(* IEC 61131-3 sources: CodesysTest/alpha/export (part 5) *)

(* ---- MotorizedSealFlattenersFB.st ---- *)
FUNCTION_BLOCK MotorizedSealFlattenersFB EXTENDS BaseComponentFB IMPLEMENTS IComponentStatus
VAR_INPUT
    {warning 'TODO: Make a struct for some of these - too many inputs'}
	sealFlattenersVerticalAxis : ICylinder();
    clearanceOffset : REAL := 0.75;        // Clearance Offset in inches
    inSetpoint : REAL := 1.25;            // In setpoint in inches
    outSetpoint : REAL := 17.7;            // Out (sealing) setpoint in inches
    bagHoldingSetpoint : REAL := 17;    // Bag holding setpoint in inches
    clearanceSpeed : INT := 3000;        // Speed to move in clearance move
    moveInSpeed : INT := 3000;            // Speed to move in in move
    moveOutSpeed : INT := 1000;            // Speed to move in out move
    moveBagHoldingSpeed : INT := 10000;    // Speed to move in bag holding move
    fingersUpSetpoint : REAL := 0;     // Fingers Up setpoint in inches
    fingersDownSetpoint : REAL := 1.1; // Fingers down setpoint in inches
    moveFingersSpeed : INT := 2000;        // Speed to move fingers
    horizontalAxisAccel : INT := 1000;    // Accel setpoint for horizontal axis
    horizontalAxisDecel : INT := 1000;    // Decel Setpoint for horizontal axis
    verticalAxisAccel : INT := 150;    // Accel setpoint for vertical axis
    verticalAxisDecel : INT := 150;    // Decel Setpoint for vertical axis
    testMovePB : BOOL;
    testMoveSP : REAL;
    stopPB : BOOL;
    startPB : BOOL;
    nextSeqPB : BOOL;
    delay : TON := (PT:= T#300MS);
	fingersDownDelay : Standard.TON := (PT := T#200MS);

	manualPosSetpoint : REAL;

END_VAR
VAR_IN_OUT
	jogIn : BOOL;
	jogOut : BOOL;
	raiseService : BOOL;
	lowerService : BOOL;
	moveToManualSetpoint : BOOL;
END_VAR
VAR_OUTPUT
    state : SEAL_FLATTENER_STATES;
END_VAR
VAR
    //pressureBarMotor : FB_FestoMotor();
    //sealFlattenersVerticalAxisMotor : FB_AppliedMotionStepServoRTU();
	jogInONS: FB_ONS;
	jogOutONS: FB_ONS;
	jogSpeed : INT := 100;
    sealFlattenersHorizontalAxisMotor : FB_AppliedMotionStepServoEIPBaseQX();
	defaultCurrentMSF : DINT := 150;
	outCurrentMSF : DINT := 150;
	bagHoldingCurrentMSF : DINT := 85;
    enableMotorizedSealFlattenersONS : R_TRIG();
    _amMoveOut : BOOL;                // Auto mode move out command
	_amMoveIn : BOOL;
    _amMoveClearance : BOOL;            // Auto mode move Clearance command
    _amMoveInToBagHolding : BOOL;    // Auto mode move in then bag holding command
END_VAR

//    Function Block:  MotorizedSealFlattenersFB
//    Description: State machine and motor management for motorized seal flateners
//    Currently, this code requires one to use the Oriental drive with pre-programmed
//    sequence for the horizontal axis
//    Created by: Ben Hess
//    Created Date: Friday, April 6, 2018
SUPER^();
// Setup and execute 2 motor axis'

// Temporary delay between states for testing
fingersDownDelay();
delay();
jogInONS(CLK := jogIn);
jogOutONS(CLK := jogOut);
IF autoModeSelected THEN
    delay.PT := T#300MS;
ELSE
    delay.PT := T#750MS;
END_IF

outSetpoint := HMIData.bagWidth + 0.2;
bagHoldingSetpoint := HMIData.bagWidth;

// Setup the vertical axis motor
sealFlattenersVerticalAxis.Execute();

// Setup the horizontal axis motor
(*
sealFlattenersHorizontalAxisMotor(modbusInBuffer := OrientalMotorModbusRead,
                stepsPerInchSetpoint := 125,
                reversePolarity := FALSE,
                operatingCurrentDefault := 500,
                modbusCommandOutBuffer := OrientalMotorCommandWrites,
                modbusParametersOutBuffer := OrientalMotorParameterWrites,
                triggerCommandWrite => OrientalMotorTriggerCommandWrite,
                triggerParameterWrite => OrientalMotorTriggerParameterWrite);
sealFlattenersHorizontalAxisMotor.Execute();
*)

sealFlattenersHorizontalAxisMotor(ptrEIPInputs := ADR(sealFlattenerHorizontalMotorInputs),
                ptrEIPOutputs := ADR(sealFlattenerHorizontalMotorOutputs),
                stepsPerInchSetpoint := Globals.STEPS_PER_INCH_SEAL_FLATTENER_HORIZONTAL_AXIS_MOTOR,
                faultHandler := PRG_Bagger.faultHandler,
				reversePolarity := TRUE,
				defaultCurrentSetpoint := defaultCurrentMSF,
				commFail := MSFMotor.udiState <> 4,
				isHomable := TRUE);

sealFlattenersHorizontalAxisMotor.Execute();

//Report as ready if mode is auto and we're not faulted
_ready := (_mode = DEVICE_MODES.Auto) AND NOT (state = SEAL_FLATTENER_STATES.Fault);

enableMotorizedSealFlattenersONS(CLK := enable);
IF stopPB THEN
    sealFlattenersHorizontalAxisMotor.Stop();
    stopPB := FALSE;
END_IF

IF startPB AND semiAutoModeSelected THEN
    //sealFlattenersHorizontalAxisMotor.StartOperation();
    startPB := FALSE;
END_IF

IF nextSeqPB THEN
    //sealFlattenersHorizontalAxisMotor.NextSequence();
    nextSeqPB := FALSE;
END_IF

IF testMovePB THEN
    sealFlattenersHorizontalAxisMotor.MoveToPosition(position := (testMoveSP), acceleration := 100, deceleration := 100, velocity := 600);
    testMovePB := FALSE;
END_IF

IF enableONS.Q OR resetONS.Q THEN
    state := SEAL_FLATTENER_STATES.Idle;
	sealFlattenersHorizontalAxisMotor.Reset();
	_reset := FALSE;
	ClearCommands();
END_IF

IF NOT enable THEN
    state := SEAL_FLATTENER_STATES.Fault;
END_IF

// State amchine for motorized seal flatteners
CASE state OF

    SEAL_FLATTENER_STATES.Idle :                                    //If enabled move to out
                                                                    IF enable AND semiAutoModeSelected OR (autoModeSelected AND _amMoveOut) THEN
                                                                        state := SEAL_FLATTENER_STATES.MoveFlattenersOut;
                                                                        ClearCommands();
                                                                    END_IF

																	IF enable AND autoModeSelected AND _amMoveIn OR _amMoveInToBagHolding THEN
																	//IF enable AND autoModeSelected AND _amMoveIn THEN
																		sealFlattenersVerticalAxis.Retract();
																		state := SEAL_FLATTENER_STATES.MoveFlattenersIn;
																		ClearCommands();
																	END_IF

																	IF jogInONS.OSR THEN
																		sealFlattenersHorizontalAxisMotor.MoveDistance(distance := -18,
																									acceleration := horizontalAxisAccel,
																									deceleration := horizontalAxisDecel,
																									velocity := jogSpeed);
																	ELSIF jogOutONS.OSR THEN
																		sealFlattenersHorizontalAxisMotor.MoveDistance(distance := 18,
																									acceleration := horizontalAxisAccel,
																									deceleration := horizontalAxisDecel,
																									velocity := jogSpeed);
																	ELSIF jogInONS.OSF OR jogOutONS.OSF THEN
																		sealFlattenersHorizontalAxisMotor.Stop();
																	END_IF

																	IF raiseService THEN
																		sealFlattenersVerticalAxis.Retract();
																		raiseService := FALSE;
																	ELSIF lowerService THEN
																		sealFlattenersVerticalAxis.Extend();
																		lowerService := FALSE;
																	END_IF

																	IF moveToManualSetpoint THEN
																		sealFlattenersHorizontalAxisMotor.MoveToPosition(position := manualPosSetpoint,
																									acceleration := horizontalAxisAccel,
																									deceleration := horizontalAxisDecel,
																									velocity := moveFingersSpeed);
																		moveToManualSetpoint := FALSE;
																	END_IF

    SEAL_FLATTENER_STATES.MoveFlattenersOut :                        // Move flatteners to out position

                                                                    //sealFlattenersHorizontalAxisMotor.StartOperation();
                                                                    sealFlattenersHorizontalAxisMotor.MoveToPositionTorque(position := outSetpoint,
                                                                                                                        acceleration := horizontalAxisAccel,
                                                                                                                        deceleration := horizontalAxisDecel,
                                                                                                                        velocity := moveOutSpeed,
																														current := outCurrentMSF);
                                                                    state := SEAL_FLATTENER_STATES.MovingFlattenersOut;

    SEAL_FLATTENER_STATES.MovingFlattenersOut :                        //
                                                                    delay.IN := TRUE;
                                                                    IF delay.Q THEN
																		IF sealFlattenersHorizontalAxisMotor.CommandAcknowledged AND sealFlattenersHorizontalAxisMotor.CurrentPosition >= (bagHoldingSetpoint - 1.5) THEN
																			state := SEAL_FLATTENER_STATES.MovedFlattenersOut;
                                                                        	delay.IN := FALSE;
																		END_IF
                                                                    END_IF

    SEAL_FLATTENER_STATES.MovedFlattenersOut :                        // Move flatteners to clearance position state
                                                                    IF enable AND semiAutoModeSelected OR (autoModeSelected AND _amMoveClearance) THEN
                                                                        state := SEAL_FLATTENER_STATES.MoveFlattenersUpAndToClearance;
                                                                        ClearCommands();
                                                                    END_IF

    SEAL_FLATTENER_STATES.MoveFlattenersUpAndToClearance :                // Move flatteners to clearance position

                                                                    //sealFlattenersHorizontalAxisMotor.NextSequence();
                                                                    sealFlattenersHorizontalAxisMotor.MoveToPosition(position := (outSetpoint - clearanceOffset),
                                                                                                                        acceleration := horizontalAxisAccel,
                                                                                                                        deceleration := horizontalAxisDecel,
                                                                                                                        velocity := moveOutSpeed);
                                                                   	sealFlattenersVerticalAxis.Retract();
                                                                    state := SEAL_FLATTENER_STATES.MovingFlattenersUpAndToClearance;

    SEAL_FLATTENER_STATES.MovingFlattenersUpAndToClearance :        delay.IN := TRUE;
                                                                    IF delay.Q THEN
																		IF sealFlattenersHorizontalAxisMotor.CommandAcknowledged AND sealFlattenersHorizontalAxisMotor.InPosition THEN
																			state := SEAL_FLATTENER_STATES.MovedFlattenersUpAndToClearance;
                                                                        	delay.IN := FALSE;
																		END_IF
                                                                    END_IF

    SEAL_FLATTENER_STATES.MovedFlattenersUpAndToClearance :                // Move flatteners to up state
                                                                    IF enable AND semiAutoModeSelected OR (autoModeSelected AND (_amMoveInToBagHolding OR _amMoveIn)) THEN
                                                                        state := SEAL_FLATTENER_STATES.MoveFlattenersIn;
                                                                        //ClearCommands();
                                                                    END_IF

    SEAL_FLATTENER_STATES.MoveFlattenersIn :                        // Move flatteners up and in
                                                                    //sealFlattenersHorizontalAxisMotor.NextSequence();
                                                                    sealFlattenersHorizontalAxisMotor.MoveToPosition(position := inSetpoint,
                                                                                                                        acceleration := horizontalAxisAccel,
                                                                                                                        deceleration := horizontalAxisDecel,
                                                                                                                        velocity := moveInSpeed);
                                                                    state := SEAL_FLATTENER_STATES.MovingFlattenersIn;

    SEAL_FLATTENER_STATES.MovingFlattenersIn :                        // If we did that command well move on
                                                                        delay.IN := TRUE;
                                                                        IF delay.Q THEN
																			IF sealFlattenersHorizontalAxisMotor.CommandAcknowledged AND sealFlattenersHorizontalAxisMotor.InPosition THEN
																				state := SEAL_FLATTENER_STATES.MovedFlattenersIn;
                                                                           		delay.IN := FALSE;
																			END_IF
                                                                        END_IF

    SEAL_FLATTENER_STATES.MovedFlattenersIn :                        // Now that we're up and in move to down and 4 corners/bag holding
                                                                    IF enable AND semiAutoModeSelected OR (autoModeSelected AND _amMoveInToBagHolding) THEN
                                                                        state := SEAL_FLATTENER_STATES.MoveFlattenersDown;
                                                                        ClearCommands();
                                                                    END_IF

    SEAL_FLATTENER_STATES.MoveFlattenersDown :            // Do moves for down and bag holding

                                                                        sealFlattenersVerticalAxis.Extend();

                                                                        state := SEAL_FLATTENER_STATES.MovingFlattenersDown;

    SEAL_FLATTENER_STATES.MovingFlattenersDown :
                                                                        //IF sealFlattenersVerticalAxis.CommandAcknowledged AND sealFlattenersVerticalAxis.InPosition THEN
                                                                       	fingersDownDelay.IN := TRUE;
																	  	IF fingersDownDelay.Q THEN
																			state := SEAL_FLATTENER_STATES.MovedFlattenersDown;
																			fingersDownDelay.IN := FALSE;
																		END_IF

                                                                        //END_IF

    SEAL_FLATTENER_STATES.MovedFlattenersDown :            state := SEAL_FLATTENER_STATES.MoveFlattenersToBagHolding;

    SEAL_FLATTENER_STATES.MoveFlattenersToBagHolding :            // Do moves for down and bag holding
                                                                        //sealFlattenersHorizontalAxisMotor.NextSequence();
                                                                        sealFlattenersHorizontalAxisMotor.MoveToPositionTorque(position := bagHoldingSetpoint,
                                                                                                                        acceleration := horizontalAxisAccel,
                                                                                                                        deceleration := horizontalAxisDecel,
                                                                                                                        velocity := moveBagHoldingSpeed,
																														current := bagHoldingCurrentMSF);
                                                                        state := SEAL_FLATTENER_STATES.MovingFlattenersToBagHolding;

    SEAL_FLATTENER_STATES.MovingFlattenersToBagHolding :            delay.IN := TRUE;
                                                                        IF delay.Q THEN
																			IF sealFlattenersHorizontalAxisMotor.CommandAcknowledged THEN
																				state := SEAL_FLATTENER_STATES.MovedFlattenersToBagHolding;
                                                                            	delay.IN := FALSE;
																			END_IF
                                                                        END_IF

    SEAL_FLATTENER_STATES.MovedFlattenersToBagHolding :            state := SEAL_FLATTENER_STATES.Idle;
																		HMIData.motorizedSealFlattenerCycles.Increment();
                                                                        Globals.motorizedSealFlattenersCount := Globals.motorizedSealFlattenersCount +1;
                                                                        Globals.sealFlattenerFingersCount := Globals.sealFlattenerFingersCount +1;
    SEAL_FLATTENER_STATES.Ready :
    SEAL_FLATTENER_STATES.Fault :
END_CASE

METHOD PRIVATE ClearCommands
VAR_INPUT
END_VAR

// Clear all commands from auto mode
_amMoveOut := FALSE;
_amMoveClearance := FALSE;
_amMoveInToBagHolding := FALSE;
_amMoveIn := FALSE;

PROPERTY Ready : BOOL

METHOD AutoMoveOut
VAR_INPUT
END_VAR

_amMoveOut := TRUE;

PROPERTY Mode : DEVICE_MODES

METHOD AutoMoveToClearance
VAR_INPUT
END_VAR

_amMoveClearance := TRUE;

METHOD AutoMoveToBagHolding
VAR_INPUT
END_VAR

_amMoveInToBagHolding := TRUE;

METHOD AutoMoveIn : BOOL
VAR_INPUT
END_VAR

_amMoveIn := TRUE;

(* ---- MotorizedSealFlattenersFB_BagFeed.st ---- *)
FUNCTION_BLOCK MotorizedSealFlattenersFB_BagFeed EXTENDS BaseComponentFB IMPLEMENTS IComponentStatus
VAR_INPUT
    {warning 'TODO: Make a struct for some of these - too many inputs'}
	sealFlattenersVerticalAxis : ICylinder();
    clearanceOffset : REAL := 2.0;        // Clearance Offset in inches
	bagFeedPosition : REAL;
    inSetpoint : REAL := 1.25;            // In setpoint in inches
    outSetpoint : REAL := 17.7;            // Out (sealing) setpoint in inches
    bagHoldingSetpoint : REAL := 17;    // Bag holding setpoint in inches
    clearanceSpeed : INT := 3000;        // Speed to move in clearance move
    moveInSpeed : INT := 3000;            // Speed to move in in move
    moveOutSpeed : INT := 1000;            // Speed to move in out move
    moveBagHoldingSpeed : INT := 1000;    // Speed to move in bag holding move
    fingersUpSetpoint : REAL := 0;     // Fingers Up setpoint in inches
    fingersDownSetpoint : REAL := 1.1; // Fingers down setpoint in inches
    moveFingersSpeed : INT := 2000;        // Speed to move fingers
    horizontalAxisAccel : INT := 1000;    // Accel setpoint for horizontal axis
    horizontalAxisDecel : INT := 1000;    // Decel Setpoint for horizontal axis
    verticalAxisAccel : INT := 150;    // Accel setpoint for vertical axis
    verticalAxisDecel : INT := 150;    // Decel Setpoint for vertical axis
    testMovePB : BOOL;
    testMoveSP : REAL;
    stopPB : BOOL;
    startPB : BOOL;
    nextSeqPB : BOOL;
    delay : TON := (PT:= T#300MS);
	fingersDownDelay : Standard.TON := (PT := T#200MS);

	manualPosSetpoint : REAL;

END_VAR
VAR_IN_OUT
	jogIn : BOOL;
	jogOut : BOOL;
	raiseService : BOOL;
	lowerService : BOOL;
	moveToManualSetpoint : BOOL;
END_VAR
VAR_OUTPUT
    state : SEAL_FLATTENER_STATES;
END_VAR
VAR
    //pressureBarMotor : FB_FestoMotor();
    //sealFlattenersVerticalAxisMotor : FB_AppliedMotionStepServoRTU();
	jogInONS: FB_ONS;
	jogOutONS: FB_ONS;
	jogSpeed : INT := 100;
    sealFlattenersHorizontalAxisMotor : FB_AppliedMotionStepServoEIPBaseQX();
	defaultCurrentMSF : DINT := 150;
	outCurrentMSF : DINT := 150;
	bagHoldingCurrentMSF : DINT := 85;
    enableMotorizedSealFlattenersONS : R_TRIG();
	bagDropDelay : Standard.TON := (PT := T#1S);
    _amMoveOut : BOOL;                // Auto mode move out command
	_amMoveIn : BOOL;
    _amMoveClearance : BOOL;            // Auto mode move Clearance command
    _amMoveInToBagHolding : BOOL;    // Auto mode move in then bag holding command
END_VAR

//    Function Block:  MotorizedSealFlattenersFB
//    Description: State machine and motor management for motorized seal flateners
//    Currently, this code requires one to use the Oriental drive with pre-programmed
//    sequence for the horizontal axis
//    Created by: Ben Hess
//    Created Date: Friday, April 6, 2018
SUPER^();
// Setup and execute 2 motor axis'

// Temporary delay between states for testing
fingersDownDelay();
bagDropDelay(PT := TO_TIME(HMIData.bagDropTime * 1000));
delay();
jogInONS(CLK := jogIn);
jogOutONS(CLK := jogOut);
IF autoModeSelected THEN
    delay.PT := T#300MS;
ELSE
    delay.PT := T#750MS;
END_IF

outSetpoint := HMIData.bagWidth + 0.2;
bagHoldingSetpoint := HMIData.bagWidth;

// Setup the vertical axis motor
sealFlattenersVerticalAxis.Execute();

// Setup the horizontal axis motor
(*
sealFlattenersHorizontalAxisMotor(modbusInBuffer := OrientalMotorModbusRead,
                stepsPerInchSetpoint := 125,
                reversePolarity := FALSE,
                operatingCurrentDefault := 500,
                modbusCommandOutBuffer := OrientalMotorCommandWrites,
                modbusParametersOutBuffer := OrientalMotorParameterWrites,
                triggerCommandWrite => OrientalMotorTriggerCommandWrite,
                triggerParameterWrite => OrientalMotorTriggerParameterWrite);
sealFlattenersHorizontalAxisMotor.Execute();
*)

sealFlattenersHorizontalAxisMotor(ptrEIPInputs := ADR(sealFlattenerHorizontalMotorInputs),
                ptrEIPOutputs := ADR(sealFlattenerHorizontalMotorOutputs),
                stepsPerInchSetpoint := Globals.STEPS_PER_INCH_SEAL_FLATTENER_HORIZONTAL_AXIS_MOTOR,
                faultHandler := PRG_Bagger.faultHandler,
				reversePolarity := TRUE,
				defaultCurrentSetpoint := defaultCurrentMSF,
				commFail := MSFMotor.udiState <> 4,
				isHomable := TRUE);

sealFlattenersHorizontalAxisMotor.Execute();

//Report as ready if mode is auto and we're not faulted
_ready := (_mode = DEVICE_MODES.Auto) AND NOT (state = SEAL_FLATTENER_STATES.Fault);

enableMotorizedSealFlattenersONS(CLK := enable);
IF stopPB THEN
    sealFlattenersHorizontalAxisMotor.Stop();
    stopPB := FALSE;
END_IF

IF startPB AND semiAutoModeSelected THEN
    //sealFlattenersHorizontalAxisMotor.StartOperation();
    startPB := FALSE;
END_IF

IF nextSeqPB THEN
    //sealFlattenersHorizontalAxisMotor.NextSequence();
    nextSeqPB := FALSE;
END_IF

IF testMovePB THEN
    sealFlattenersHorizontalAxisMotor.MoveToPosition(position := (testMoveSP), acceleration := 100, deceleration := 100, velocity := 600);
    testMovePB := FALSE;
END_IF

IF enableONS.Q OR resetONS.Q THEN
    state := SEAL_FLATTENER_STATES.Idle;
	sealFlattenersHorizontalAxisMotor.Reset();
	_reset := FALSE;
	bagDropDelay.IN := FALSE;
	ClearCommands();
END_IF

IF NOT enable THEN
    state := SEAL_FLATTENER_STATES.Fault;
END_IF

// State amchine for motorized seal flatteners
CASE state OF

    SEAL_FLATTENER_STATES.Idle :                                    //If enabled move to out
                                                                    IF enable AND semiAutoModeSelected OR (autoModeSelected AND _amMoveOut) THEN
                                                                        state := SEAL_FLATTENER_STATES.MoveFlattenersOut;
                                                                        ClearCommands();
                                                                    END_IF

																	IF enable AND autoModeSelected AND _amMoveIn OR _amMoveInToBagHolding THEN
																	//IF enable AND autoModeSelected AND _amMoveIn THEN
																		sealFlattenersVerticalAxis.Retract();
																		state := SEAL_FLATTENER_STATES.MoveFlattenersIn;
																		ClearCommands();
																	END_IF

																	IF jogInONS.OSR THEN
																		sealFlattenersHorizontalAxisMotor.MoveDistance(distance := -18,
																									acceleration := horizontalAxisAccel,
																									deceleration := horizontalAxisDecel,
																									velocity := jogSpeed);
																	ELSIF jogOutONS.OSR THEN
																		sealFlattenersHorizontalAxisMotor.MoveDistance(distance := 18,
																									acceleration := horizontalAxisAccel,
																									deceleration := horizontalAxisDecel,
																									velocity := jogSpeed);
																	ELSIF jogInONS.OSF OR jogOutONS.OSF THEN
																		sealFlattenersHorizontalAxisMotor.Stop();
																	END_IF

																	IF raiseService THEN
																		sealFlattenersVerticalAxis.Retract();
																		raiseService := FALSE;
																	ELSIF lowerService THEN
																		sealFlattenersVerticalAxis.Extend();
																		lowerService := FALSE;
																	END_IF

																	IF moveToManualSetpoint THEN
																		sealFlattenersHorizontalAxisMotor.MoveToPosition(position := manualPosSetpoint,
																									acceleration := horizontalAxisAccel,
																									deceleration := horizontalAxisDecel,
																									velocity := moveFingersSpeed);
																		moveToManualSetpoint := FALSE;
																	END_IF

																	bagDropDelay.IN := FALSE;

    SEAL_FLATTENER_STATES.MoveFlattenersOut :                        // Move flatteners to out position

                                                                    //sealFlattenersHorizontalAxisMotor.StartOperation();
                                                                    sealFlattenersHorizontalAxisMotor.MoveToPositionTorque(position := outSetpoint,
                                                                                                                        acceleration := horizontalAxisAccel,
                                                                                                                        deceleration := horizontalAxisDecel,
                                                                                                                        velocity := moveOutSpeed,
																														current := outCurrentMSF);
                                                                    state := SEAL_FLATTENER_STATES.MovingFlattenersOut;

    SEAL_FLATTENER_STATES.MovingFlattenersOut :                        //
                                                                    delay.IN := TRUE;
                                                                    IF delay.Q THEN
																		IF sealFlattenersHorizontalAxisMotor.CommandAcknowledged AND sealFlattenersHorizontalAxisMotor.CurrentPosition >= (bagHoldingSetpoint - 1.5) THEN
																			state := SEAL_FLATTENER_STATES.MovedFlattenersOut;
                                                                        	delay.IN := FALSE;
																		END_IF
                                                                    END_IF

    SEAL_FLATTENER_STATES.MovedFlattenersOut :                        // Move flatteners to clearance position state
                                                                    IF enable AND semiAutoModeSelected OR (autoModeSelected AND _amMoveClearance) THEN
                                                                        state := SEAL_FLATTENER_STATES.MoveFlattenersUpAndToClearance;
                                                                        ClearCommands();
                                                                    END_IF

    SEAL_FLATTENER_STATES.MoveFlattenersUpAndToClearance :                // Move flatteners to clearance position

                                                                    //sealFlattenersHorizontalAxisMotor.NextSequence();
                                                                    sealFlattenersHorizontalAxisMotor.MoveToPosition(position := (outSetpoint - clearanceOffset),
                                                                                                                        acceleration := horizontalAxisAccel,
                                                                                                                        deceleration := horizontalAxisDecel,
                                                                                                                        velocity := moveOutSpeed);
                                                                   	sealFlattenersVerticalAxis.Retract();
                                                                    state := SEAL_FLATTENER_STATES.MovingFlattenersUpAndToClearance;

    SEAL_FLATTENER_STATES.MovingFlattenersUpAndToClearance :        delay.IN := TRUE;
                                                                    IF delay.Q THEN
																		IF sealFlattenersHorizontalAxisMotor.CommandAcknowledged AND sealFlattenersHorizontalAxisMotor.InPosition THEN
																			state := SEAL_FLATTENER_STATES.MovedFlattenersUpAndToClearance;
                                                                        	delay.IN := FALSE;
																		END_IF

                                                                    END_IF

    SEAL_FLATTENER_STATES.MovedFlattenersUpAndToClearance :                // Move flatteners to up state
																	bagDropDelay.IN := TRUE;
																	IF bagDropDelay.Q THEN
																		state := SEAL_FLATTENER_STATES.MoveFlattenersToBagFeed;
																		bagDropDelay.IN := FALSE;
																	END_IF

	SEAL_FLATTENER_STATES.MoveFlattenersToBagFeed :      			// Move flatteners to out of the way of the bag for feeding
																	IF (outSetpoint + clearanceOffset) <= 18.2 THEN
																		bagFeedPosition := (outSetpoint + clearanceOffset);
																	ELSE
																		bagFeedPosition := 18.2;
																	END_IF

                                                                    sealFlattenersHorizontalAxisMotor.MoveToPosition(position := bagFeedPosition,
                                                                                                                        acceleration := horizontalAxisAccel,
                                                                                                                        deceleration := horizontalAxisDecel,
                                                                                                                        velocity := moveInSpeed);
                                                                    state := SEAL_FLATTENER_STATES.MovingFlattenersToBagFeed;

   SEAL_FLATTENER_STATES.MovingFlattenersToBagFeed :        			delay.IN := TRUE;
                                                                    IF delay.Q THEN
																		IF sealFlattenersHorizontalAxisMotor.CommandAcknowledged AND sealFlattenersHorizontalAxisMotor.InPosition THEN
																			state := SEAL_FLATTENER_STATES.MovedFlattenersToBagFeed;
                                                                        	delay.IN := FALSE;
																		END_IF
                                                                    END_IF

	SEAL_FLATTENER_STATES.MovedFlattenersToBagFeed:					       // Move flatteners to up state
                                                                    IF enable AND semiAutoModeSelected OR (autoModeSelected AND (_amMoveInToBagHolding OR _amMoveIn)) THEN
                                                                        state := SEAL_FLATTENER_STATES.MoveFlattenersIn;
                                                                        //ClearCommands();
                                                                    END_IF

    SEAL_FLATTENER_STATES.MoveFlattenersIn :                        // Move flatteners up and in
                                                                    //sealFlattenersHorizontalAxisMotor.NextSequence();
                                                                    sealFlattenersHorizontalAxisMotor.MoveToPosition(position := inSetpoint,
                                                                                                                        acceleration := horizontalAxisAccel,
                                                                                                                        deceleration := horizontalAxisDecel,
                                                                                                                        velocity := moveInSpeed);
                                                                    state := SEAL_FLATTENER_STATES.MovingFlattenersIn;

    SEAL_FLATTENER_STATES.MovingFlattenersIn :                        // If we did that command well move on
                                                                        delay.IN := TRUE;
                                                                        IF delay.Q THEN
																			IF sealFlattenersHorizontalAxisMotor.CommandAcknowledged AND sealFlattenersHorizontalAxisMotor.InPosition THEN
																				state := SEAL_FLATTENER_STATES.MovedFlattenersIn;
                                                                           		delay.IN := FALSE;
																			END_IF
                                                                        END_IF

    SEAL_FLATTENER_STATES.MovedFlattenersIn :                        // Now that we're up and in move to down and 4 corners/bag holding
                                                                    IF enable AND semiAutoModeSelected OR (autoModeSelected AND _amMoveInToBagHolding) THEN
                                                                        state := SEAL_FLATTENER_STATES.MoveFlattenersDown;
                                                                        ClearCommands();
                                                                    END_IF

    SEAL_FLATTENER_STATES.MoveFlattenersDown :            // Do moves for down and bag holding

                                                                        sealFlattenersVerticalAxis.Extend();

                                                                        state := SEAL_FLATTENER_STATES.MovingFlattenersDown;

    SEAL_FLATTENER_STATES.MovingFlattenersDown :
                                                                        //IF sealFlattenersVerticalAxis.CommandAcknowledged AND sealFlattenersVerticalAxis.InPosition THEN
                                                                       	fingersDownDelay.IN := TRUE;
																	  	IF fingersDownDelay.Q THEN
																			state := SEAL_FLATTENER_STATES.MovedFlattenersDown;
																			fingersDownDelay.IN := FALSE;
																		END_IF

                                                                        //END_IF

    SEAL_FLATTENER_STATES.MovedFlattenersDown :            state := SEAL_FLATTENER_STATES.MoveFlattenersToBagHolding;

    SEAL_FLATTENER_STATES.MoveFlattenersToBagHolding :            // Do moves for down and bag holding
                                                                        //sealFlattenersHorizontalAxisMotor.NextSequence();
                                                                        sealFlattenersHorizontalAxisMotor.MoveToPositionTorque(position := bagHoldingSetpoint,
                                                                                                                        acceleration := horizontalAxisAccel,
                                                                                                                        deceleration := horizontalAxisDecel,
                                                                                                                        velocity := moveBagHoldingSpeed,
																														current := bagHoldingCurrentMSF);
                                                                        state := SEAL_FLATTENER_STATES.MovingFlattenersToBagHolding;

    SEAL_FLATTENER_STATES.MovingFlattenersToBagHolding :            delay.IN := TRUE;
                                                                        IF delay.Q THEN
																			IF sealFlattenersHorizontalAxisMotor.CommandAcknowledged THEN
																				state := SEAL_FLATTENER_STATES.MovedFlattenersToBagHolding;
                                                                            	delay.IN := FALSE;
																			END_IF
                                                                        END_IF

    SEAL_FLATTENER_STATES.MovedFlattenersToBagHolding :            state := SEAL_FLATTENER_STATES.Idle;
																		HMIData.motorizedSealFlattenerCycles.Increment();
                                                                        Globals.motorizedSealFlattenersCount := Globals.motorizedSealFlattenersCount +1;
                                                                        Globals.sealFlattenerFingersCount := Globals.sealFlattenerFingersCount +1;
    SEAL_FLATTENER_STATES.Ready :
    SEAL_FLATTENER_STATES.Fault :
END_CASE

METHOD PRIVATE ClearCommands
VAR_INPUT
END_VAR

// Clear all commands from auto mode
_amMoveOut := FALSE;
_amMoveClearance := FALSE;
_amMoveInToBagHolding := FALSE;
_amMoveIn := FALSE;

PROPERTY Ready : BOOL

METHOD AutoMoveOut
VAR_INPUT
END_VAR

_amMoveOut := TRUE;

PROPERTY Mode : DEVICE_MODES

METHOD AutoMoveToClearance
VAR_INPUT
END_VAR

_amMoveClearance := TRUE;

METHOD AutoMoveToBagHolding
VAR_INPUT
END_VAR

_amMoveInToBagHolding := TRUE;

METHOD AutoMoveIn : BOOL
VAR_INPUT
END_VAR

_amMoveIn := TRUE;

(* ---- MurrIOFB.st ---- *)
FUNCTION_BLOCK MurrIOFB EXTENDS BaseComponentFB IMPLEMENTS IComponentStatus
VAR_INPUT
	headNodeEnabled : BOOL;
	guardNodeEnabled : BOOL;
	printerNodeEnabled : BOOL;
	dischargeNodeEnabled : BOOL;
	auxIONodeEnabled : BOOL;
	configVersion : CONFIG_VERSIONS;
	MachineOptionsManagementOutputs : POINTER TO BYTE;
	SystemStatusInputs : POINTER TO BYTE;
END_VAR
VAR_OUTPUT

END_VAR
VAR
	systemStatusINT : INT;
	systemStatusState : MURR_SYSTEM_STATES;
	toggleConfig : OSCAT_BASIC.GEN_SQ;
	MOMConfigLast : BYTE;
END_VAR

VAR_IN_OUT

END_VAR

//    Function Block: MurrIOFB
//    Description: Alarms, faults, configuration of the Murr Cube67+ Bus Node
//    Created by: Ben Hess
//    Created Date: October 16th, 2019
SUPER^();
toggleConfig(PT := T#20MS);
IF MachineOptionsManagementOutputs = 0 OR SystemStatusInputs = 0 THEN
	RETURN;
END_IF
// MOM config - MOM bits are counted from Slot 001 to 4xx and are counted based on the "Maximium" configuration hard coded in the bus master
// Here we can select which verison of code we have in order to utilize MOM correctly if we add additional modules in the future.
CASE configVersion OF
	CONFIG_VERSIONS.V_1_1 :		//
									MachineOptionsManagementOutputs[0].0 := NOT headNodeEnabled;
									MachineOptionsManagementOutputs[0].1 := NOT guardNodeEnabled;
									MachineOptionsManagementOutputs[0].2 := NOT dischargeNodeEnabled;
									MachineOptionsManagementOutputs[0].3 := NOT printerNodeEnabled;
									MachineOptionsManagementOutputs[0].4 := FALSE;

	CONFIG_VERSIONS.V_1_2 : 		// Added aux IO to this version
									MachineOptionsManagementOutputs[0].0 := NOT headNodeEnabled;
									MachineOptionsManagementOutputs[0].1 := NOT guardNodeEnabled;
									MachineOptionsManagementOutputs[0].2 := NOT auxIONodeEnabled;
									MachineOptionsManagementOutputs[0].3 := NOT dischargeNodeEnabled;
									MachineOptionsManagementOutputs[0].4 := NOT printerNodeEnabled;
END_CASE

// Run config if IO bus node is waiting on config
systemStatusINT := SystemStatusInputs^;
systemStatusState := systemStatusINT;

CASE systemStatusState OF
	//MURR_SYSTEM_STATES.Internal_Comm_OK:			// If config changes here, send it down
// 													IF MachineOptionsManagementOutputs[0] <> MOMConfigLast THEN
// 														MachineOptionsManagementOutputs[4].0 := TRUE;
// 														MOMConfigLast := MachineOptionsManagementOutputs[0];
// 													END_IF

	MURR_SYSTEM_STATES.Waiting_For_MOM: 			// Bit 32 is Configure Node
													MachineOptionsManagementOutputs[4].0 := TRUE;

	MURR_SYSTEM_STATES.Configuring_MOM : 			//
													MachineOptionsManagementOutputs[4].0 := FALSE;

ELSE
	MachineOptionsManagementOutputs[4].0 := FALSE;
END_CASE

PROPERTY Mode : DEVICE_MODES

PROPERTY Ready : BOOL

(* ---- PickAndPlaceFB.st ---- *)
FUNCTION_BLOCK PickAndPlaceFB EXTENDS BaseComponentFB
VAR_INPUT
	XAxisMotor : IPositionableMotor;	// X Axis Motor
	YAxisMotor : IPositionableMotor;	// Y Axis Motor
	ZAxisMotor : IPositionableMotor;	// Z Axis Motor
END_VAR
VAR_OUTPUT
	state : VACUUM_PICKER_STATES;	 //State indication
END_VAR
VAR

	accel : INT := 2000;
	decel : INT := 2000;
	velo : INT := 2000;
	zVelo : INT := 12000;
END_VAR

//	Function Block: PickAndPlaceFB
//	Description: This provides the methods and state machine to operate the Vacuum Head pick and place machine
//
//	Created by: Ben Hess
//	Created Date: Friday, June 1, 2018

// Run the base FB
SUPER^();

// Set up the 3 motors.

// X Axis moves out and in relative to the machine. Out is 0in, max in is 7.5in.

IF enableONS.Q THEN
    IF _mode = DEVICE_MODES.Manual THEN
        state := VACUUM_PICKER_STATES.Manual;
    ELSE
        state := VACUUM_PICKER_STATES.Ready;
    END_IF
END_IF

IF NOT enable THEN
    state := VACUUM_PICKER_STATES.Idle;
END_IF

_ready := (_mode = DEVICE_MODES.Auto) AND NOT (state = VACUUM_PICKER_STATES.Fault);

CASE state OF
	VACUUM_PICKER_STATES.Idle :
	VACUUM_PICKER_STATES.Home :								// Move everything to home position
															XAxisMotor.MoveToPosition(6, accel,decel,velo);
															YAxisMotor.MoveToPosition(15, accel,decel,velo);
															ZAxisMotor.MoveToPosition(1, accel,decel,zVelo);
															state := VACUUM_PICKER_STATES.Homing;

	VACUUM_PICKER_STATES.Homing :							// Move on if all motors report ready
															IF XAxisMotor.CurrentPosition = 6
																AND YAxisMotor.CurrentPosition = 15
																AND ZAxisMotor.CurrentPosition = 1 THEN
																	state := VACUUM_PICKER_STATES.Homed;
															END_IF

	VACUUM_PICKER_STATES.Homed :							//
															state :=VACUUM_PICKER_STATES.XAxisMoveIn;

	VACUUM_PICKER_STATES.XAxisMoveIn :						// Move XAxis in
															XAxisMotor.MoveToPosition(0,accel,decel,velo);
															state := VACUUM_PICKER_STATES.XAxisMovingIn;

	VACUUM_PICKER_STATES.XAxisMovingIn :					//
															IF XAxisMotor.CurrentPosition = 0 THEN
																state := VACUUM_PICKER_STATES.XaxisMovedIn;
															END_IF

	VACUUM_PICKER_STATES.XaxisMovedIn :						//
															state := VACUUM_PICKER_STATES.VacuumTurnOn;

	VACUUM_PICKER_STATES.VacuumTurnOn :						//
															state := VACUUM_PICKER_STATES.VacuumHeadDown;

	VACUUM_PICKER_STATES.VacuumHeadDown :					//
															ZAxisMotor.MoveToPosition(150,accel,decel,zVelo);
															state := VACUUM_PICKER_STATES.YAxisMoveDown;

	VACUUM_PICKER_STATES.YAxisMoveDown :					//
															YAxisMotor.MoveToPosition(1,accel,decel,velo);
															state := VACUUM_PICKER_STATES.VacuumHeadAndYAxisMovingDown;

	VACUUM_PICKER_STATES.VacuumHeadAndYAxisMovingDown :		//
															IF YAxisMotor.CurrentPosition = 1
																AND ZAxisMotor.CurrentPosition = 150 THEN
																state := VACUUM_PICKER_STATES.VacuumHeadAndYAxisMovedDown;
															END_IF

	VACUUM_PICKER_STATES.VacuumHeadAndYAxisMovedDown :		//
															state := VACUUM_PICKER_STATES.VacuumTurnOff;

	VACUUM_PICKER_STATES.VacuumTurnOff :					//
															state := VACUUM_PICKER_STATES.ConveyorTurnOn;

	VACUUM_PICKER_STATES.ConveyorTurnOn :					//
															state := VACUUM_PICKER_STATES.ConveyorMoving;

	VACUUM_PICKER_STATES.ConveyorMoving :					//
															state := VACUUM_PICKER_STATES.ConveyorDone;

	VACUUM_PICKER_STATES.ConveyorDone :						//
															state := VACUUM_PICKER_STATES.Ready;

	VACUUM_PICKER_STATES.Fault :							//

	VACUUM_PICKER_STATES.Ready :							IF semiAutoModeSelected THEN
																state := VACUUM_PICKER_STATES.Home;
															END_IF
	VACUUM_PICKER_STATES.Manual :
END_CASE

(* ---- PneumaticPressureBarFB.st ---- *)
FUNCTION_BLOCK PneumaticPressureBarFB
VAR_INPUT
    enable : BOOL;                    // Enable Pneumatic pressure bar
    sealBarEnable : BOOL;            //Enable seal bar
    bagOpenFingersEnable : BOOL;        //Enable bag open fingers
	iPressureBarRetracted : BOOL;
	iPressureBarExtended : BOOL;
END_VAR
VAR_OUTPUT
    state : PRESSURE_BAR_STATES;     //Jaw State
	oPositionBagOpenFingersToRelease : BOOL;
	oExtendSealBar : BOOL;
	oExtendCylinder : BOOL;
	oRetractCylinder : BOOL;
END_VAR
VAR
    _mode : DEVICE_MODES;            // Auto-SemiAuto-Manual
    _ready : BOOL;                    // Ready to be controlled
    _amOpenJaw : BOOL;    // Auto Mode Open Jaw Command
    _amCloseJaw : BOOL;     // Auto Mode Close Jaw Command
	_amSealBag : BOOL;		// Auto mode seal bag command
    enableONS : R_TRIG; //Enable One Shot
    //autoModeSelect : BOOL;            //Auto Mode Selection (Timers)
    startCyclePB : BOOL;                //Start Cycle
    stopCyclePB : BOOL;                //Stop Cycle
    manualExtendHighPressurePB : BOOL;            //Manually Extend Cylinder High Pressure
    manualExtendLowPressurePB : BOOL;            //Manually Extend Cylinder Low Pressure
    manualRetractPB : BOOL;            //Manually Retract Cylinder
    manualExhaustPB : BOOL;            //Manually Echaust Cylinder
    timerExtendedDebounce : TON;            //Timer for extend delay
    timerExtendDwell : TON;            //Timer for extend dwell after extended
    timerRetractedDebounce : TON;        //Timer for retract delay
    timerRetractDwell : TON;        //Timer for retract dwell after extended
    timerSealDwell : TON;            //Timer for seal dwell
    extendDelaySP : INT := 50;    //Extend delay SP
    extendDwellSP : INT := 300;    //Extend dwell SP
    retractDelaySP : INT := 50;        //Retract delay SP
    retractDwellSP : INT := 750;    //Retract dwell SP
    incrementCount : R_TRIG();

    bagOpenFingersReleaseDelay : TON := (PT := T#100MS);                //Delay to open Bag Open Fingers after closing pressure bar
    bagOpenFingersGrabDelay : TON := (PT := T#100MS);                //Delay to close Bag Open Fingers after opening pressure bar
    bagOpenFingers : BagOpenFingersFB();
    openingBag : BOOL;                        //Opening bag flag for bag open fingers
    incrementSealBarCountONS : Standard.R_TRIG;
    incrementBagOpenFinersONS : Standard.R_TRIG;
    autoModeSelected : BOOL;
    semiAutoModeSelected : BOOL;
    manualModeSelected : BOOL;
END_VAR
VAR_IN_OUT

END_VAR
//    Function Block: Cylinder
//    Description: This program moves a jaw cylinder back and forth
//    Created by: Ben Hess
//    Created Date: January 16th, 2017

bagOpenFingers(releaseOutput => oPositionBagOpenFingersToRelease);

//Stop the auto cycle if button pressed or coming out of auto mode or moving the servo.
IF stopCyclePB OR NOT (_mode = DEVICE_MODES.SemiAuto) THEN
    startCyclePB := FALSE;
END_IF

autoModeSelected := (_mode = DEVICE_MODES.Auto);
semiAutoModeSelected := (_mode = DEVICE_MODES.SemiAuto);
manualModeSelected := (_mode = DEVICE_MODES.Manual);

timerExtendedDebounce(PT := INT_TO_TIME(extendDelaySP));
timerExtendDwell(PT := INT_TO_TIME(extendDwellSP));
timerRetractedDebounce(PT := INT_TO_TIME(retractDelaySP));
timerRetractDwell(PT := INT_TO_TIME(retractDwellSP));
bagOpenFingersReleaseDelay();
bagOpenFingersGrabDelay();

//Go to idle when enabled
enableONS(CLK := enable);
IF enableONS.Q THEN
    state := PRESSURE_BAR_STATES.Idle;
END_IF

IF NOT enable THEN
    state := PRESSURE_BAR_STATES.Idle;
END_IF

_ready := (_mode = DEVICE_MODES.Auto) AND NOT (state = PRESSURE_BAR_STATES.Fault);

CASE state OF

    PRESSURE_BAR_STATES.Idle :                //Initial state
                                    IF (semiAutoModeSelected AND startCyclePB) OR (autoModeSelected AND _amOpenJaw) THEN
                                        state := PRESSURE_BAR_STATES.OpenJaw;
                                        _amOpenJaw := FALSE;
                                    ELSIF (autoModeSelected AND _amCloseJaw) THEN
                                        state := PRESSURE_BAR_STATES.CloseJaw;
										_amCloseJaw := FALSE;
                                    ELSIF manualModeSelected THEN
                                        state := PRESSURE_BAR_STATES.Manual;
                                    END_IF
                                    oExtendSealBar := FALSE;

    PRESSURE_BAR_STATES.OpenJaw :                //Open jaw by extending cylinder
                                    ExtendCylinderHighPressure();
                                    state := PRESSURE_BAR_STATES.OpeningJaw;

    PRESSURE_BAR_STATES.OpeningJaw :            //
                                    //This delay is a debounce for the sensors.
                                    IF iPressureBarExtended THEN
                                        timerExtendedDebounce.IN := TRUE;
                                        IF timerExtendedDebounce.Q THEN
                                            state := PRESSURE_BAR_STATES.JawOpened;
                                            timerExtendedDebounce.IN := FALSE;
                                        END_IF
                                    END_IF
                                    //If we are opening bag this cycle then grab it now
                                    bagOpenFingersGrabDelay.IN := bagOpenFingersEnable;
                                    IF bagOpenFingersGrabDelay.Q THEN
                                        bagOpenFingers.Grab();
                                        bagOpenFingersGrabDelay.IN := FALSE;
                                    END_IF

    PRESSURE_BAR_STATES.JawOpened :            //Jaw is opened.  If in semi auto mode, go to close jaw after extend dwell.
                                    IF (semiAutoModeSelected AND startCyclePB) OR (autoModeSelected AND _amCloseJaw) THEN
                                        timerExtendDwell.IN := TRUE;
                                    END_IF

                                    IF timerExtendDwell.Q  THEN
                                        state := PRESSURE_BAR_STATES.CloseJaw;
                                        _amCloseJaw := FALSE;
                                        timerExtendDwell.IN := FALSE;
                                    END_IF

    PRESSURE_BAR_STATES.CloseJaw :            //Close jaw by retracting cylinder
                                    RetractCylinder();
                                    state := PRESSURE_BAR_STATES.ClosingJaw;

    PRESSURE_BAR_STATES.ClosingJaw :            //
                                    //This delay is a debounce after the sensor is seen
                                    IF iPressureBarRetracted THEN
                                        timerRetractedDebounce.IN := TRUE;
                                        IF timerRetractedDebounce.Q THEN
                                            state := PRESSURE_BAR_STATES.JawClosed;
                                            timerRetractedDebounce.IN := FALSE;
                                        END_IF
                                    END_IF

    PRESSURE_BAR_STATES.JawClosed :            //Go to sealing if seal bar enabled, otherwise if in auto mode go to open jaw after retract dwell. Else go back to idle
                                    IF sealBarEnable THEN
                                        state := PRESSURE_BAR_STATES.Sealing;
                                    END_IF

                                    IF (semiAutoModeSelected AND startCyclePB) OR (autoModeSelected AND _amOpenJaw) THEN
                                        bagOpenFingersReleaseDelay.IN := bagOpenFingersEnable;
                                        timerRetractDwell.IN := TRUE;
                                    END_IF

                                    IF bagOpenFingersReleaseDelay.Q THEN
                                        bagOpenFingers.Release();
                                        bagOpenFingersReleaseDelay.IN := FALSE;
                                    END_IF

                                    IF timerRetractDwell.Q THEN
                                        state := PRESSURE_BAR_STATES.OpenJaw;
                                        _amOpenJaw := FALSE;
                                        timerRetractDwell.IN := FALSE;
                                    END_IF

    PRESSURE_BAR_STATES.Sealing :                //Seal sets output for seal bar after closed for a dwell setpoint  Hack for now
                                    timerRetractDwell.IN := TRUE;

                                    IF (semiAutoModeSelected OR (autoModeSelected AND _amOpenJaw)) AND timerRetractDwell.Q THEN
                                        state := PRESSURE_BAR_STATES.OpenJaw;
                                        timerRetractDwell.IN := FALSE;
                                        _amOpenJaw := FALSE;
                                    END_IF

                                    bagOpenFingersReleaseDelay.IN := bagOpenFingersEnable;
                                    IF bagOpenFingersReleaseDelay.Q THEN
                                        bagOpenFingers.Release();
                                        bagOpenFingersReleaseDelay.IN := FALSE;
                                    END_IF

                                    oExtendSealBar := TIME_TO_REAL(timerRetractDwell.ET) > (retractDwellSP * 0.1) AND TIME_TO_REAL(timerRetractDwell.ET) < (retractDwellSP * 0.8);

    PRESSURE_BAR_STATES.Manual :    IF manualExhaustPB THEN
                                        ExhaustCylinder();
                                        manualExhaustPB := FALSE;
                                    ELSIF manualRetractPB THEN
                                        RetractCylinder();
                                        manualRetractPB := FALSE;
                                    ELSIF manualExtendHighPressurePB THEN
                                        ExtendCylinderHighPressure();
                                        manualExtendHighPressurePB := FALSE;
									ELSIF manualExtendLowPressurePB THEN
                                        ExtendCylinderLowPressure();
                                        manualExtendLowPressurePB := FALSE;
                                    END_IF

    PRESSURE_BAR_STATES.Fault :

END_CASE

//Count cycles
incrementCount(CLK :=timerExtendDwell.Q);
IF incrementCount.Q THEN
    Globals.headCycleCount := Globals.headCycleCount + 1;
END_IF

incrementSealBarCountONS(CLK := oExtendSealBar);
IF incrementSealBarCountONS.Q THEN
    Globals.sealBarCount := Globals.sealBarCount + 1;
END_IF

incrementBagOpenFinersONS(CLK := oPositionBagOpenFingersToRelease);
IF incrementBagOpenFinersONS.Q THEN
    Globals.bagOpenFingersCount := Globals.bagOpenFingersCount + 1;
END_IF

METHOD AutoDoneMovingPassthrough
VAR_INPUT
END_VAR

state := PRESSURE_BAR_STATES.Idle;

METHOD AutoMovingPassthrough
VAR_INPUT
END_VAR

state := PRESSURE_BAR_STATES.Manual;

METHOD ExhaustCylinder
VAR_INPUT
END_VAR

oExtendCylinder := FALSE;
oRetractCylinder := FALSE;

PROPERTY Mode : DEVICE_MODES

PROPERTY Ready : BOOL

METHOD AutoCloseJaw
VAR_INPUT
END_VAR

_amCloseJaw := TRUE;

METHOD ExtendCylinderHighPressure
VAR_INPUT
END_VAR

oExtendCylinder := TRUE;
oRetractCylinder := FALSE;

METHOD ExtendCylinderLowPressure
VAR_INPUT
END_VAR

oExtendCylinder := TRUE;
oRetractCylinder := TRUE;

METHOD AutoOpenJaw
VAR_INPUT
END_VAR

_amOpenJaw := TRUE;

METHOD RetractCylinder
VAR_INPUT
END_VAR

oExtendCylinder := FALSE;
oRetractCylinder := TRUE;

METHOD AutoSealBag
VAR_INPUT
END_VAR

(* ---- PneumaticPressureBarFB_1.st ---- *)
FUNCTION_BLOCK PneumaticPressureBarFB_1 EXTENDS BaseComponentFB
VAR_INPUT
	iPressureBarRetracted : BOOL;
	iPressureBarExtended : BOOL;
	iPressureBarNotObstructed : BOOL;
END_VAR
VAR_OUTPUT
    state : PRESSURE_BAR_STATES;     //Jaw State
	oExtendCylinder : BOOL;
	oRetractCylinder : BOOL;
	faults : PressureBarFaultsType;
END_VAR
VAR
    _amOpenJaw : BOOL;    // Auto Mode Open Jaw Command
    _amCloseJaw : BOOL;     // Auto Mode Close Jaw Command
    startCyclePB : BOOL;                //Start Cycle
    stopCyclePB : BOOL;                //Stop Cycle
    manualExtendHighPressurePB : BOOL;            //Manually Extend Cylinder High Pressure
    manualExtendLowPressurePB : BOOL;            //Manually Extend Cylinder Low Pressure
    manualRetractPB : BOOL;            //Manually Retract Cylinder
    manualExhaustPB : BOOL;            //Manually Echaust Cylinder
    timerExtendedDebounce : TON;            //Timer for extend delay
    timerExtendDwell : TON;            //Timer for extend dwell after extended
    timerRetractedDebounce : TON;        //Timer for retract delay
    timerRetractDwell : TON;        //Timer for retract dwell after extended
    timerSealDwell : TON;            //Timer for seal dwell
	timerObsSwitchFault : Standard.TON;
    extendDelaySP : INT := 50;    //Extend delay SP
    extendDwellSP : INT := 300;    //Extend dwell SP
    retractDelaySP : INT := 50;        //Retract delay SP
    retractDwellSP : INT := 750;    //Retract dwell SP
    incrementCount : R_TRIG();
    incrementSealBarCountONS : Standard.R_TRIG;
    incrementBagOpenFinersONS : Standard.R_TRIG;
	faultTimer : Standard.TON;
END_VAR
VAR_IN_OUT
	cumulativeHeadCycleCount : DINT;
END_VAR
//    Function Block: Cylinder
//    Description: This program moves a jaw cylinder back and forth
//    Created by: Ben Hess
//    Created Date: January 16th, 2017

SUPER^();

//Stop the auto cycle if button pressed or coming out of auto mode or moving the servo.
IF stopCyclePB OR NOT (_mode = DEVICE_MODES.SemiAuto) THEN
    startCyclePB := FALSE;
END_IF

HMIData.pressureBarService.retractedFeedback := iPressureBarRetracted;
HMIData.pressureBarService.extendedFeedback := iPressureBarExtended;

autoModeSelected := (_mode = DEVICE_MODES.Auto);
semiAutoModeSelected := (_mode = DEVICE_MODES.SemiAuto);
manualModeSelected := (_mode = DEVICE_MODES.Manual);

timerExtendedDebounce(PT := INT_TO_TIME(extendDelaySP));
timerExtendDwell(PT := INT_TO_TIME(extendDwellSP));
timerRetractedDebounce(PT := INT_TO_TIME(retractDelaySP));
timerRetractDwell(PT := INT_TO_TIME(retractDwellSP));
timerObsSwitchFault(PT := T#100MS);
//Go to idle when enabled
IF enableONS.Q OR resetONS.Q THEN
    state := PRESSURE_BAR_STATES.Idle;
	_reset := FALSE;
	timerObsSwitchFault.IN := FALSE;
END_IF

IF NOT enable THEN
    state := PRESSURE_BAR_STATES.Idle;
END_IF

_ready := (_mode = DEVICE_MODES.Auto) AND NOT (state = PRESSURE_BAR_STATES.Fault);

faultTimer();

CASE state OF

    PRESSURE_BAR_STATES.Idle :                //Initial state
                                    IF (semiAutoModeSelected AND startCyclePB) OR (autoModeSelected AND _amOpenJaw) OR HMIData.pressureBarService.extendCommand THEN
                                        state := PRESSURE_BAR_STATES.OpenJaw;
                                        _amOpenJaw := FALSE;
										HMIData.pressureBarService.extendCommand := FALSE;
                                    ELSIF (autoModeSelected AND _amCloseJaw) OR HMIData.pressureBarService.retractCommand THEN
                                        state := PRESSURE_BAR_STATES.CloseJaw;
										_amCloseJaw := FALSE;
										HMIData.pressureBarService.retractCommand := FALSE;
                                    ELSIF manualModeSelected THEN
                                        state := PRESSURE_BAR_STATES.Manual;
                                    END_IF
                                    timerObsSwitchFault.IN := FALSE;

    PRESSURE_BAR_STATES.OpenJaw :                //Open jaw by extending cylinder
                                    ExtendCylinderHighPressure();
                                    state := PRESSURE_BAR_STATES.OpeningJaw;

    PRESSURE_BAR_STATES.OpeningJaw :            //
                                    //This delay is a debounce for the sensors.
                                    faultTimer.PT := T#3S;
									faultTimer.IN := TRUE;
									IF iPressureBarExtended THEN
                                        timerExtendedDebounce.IN := TRUE;
                                        IF timerExtendedDebounce.Q THEN
                                            state := PRESSURE_BAR_STATES.JawOpened;
                                            timerExtendedDebounce.IN := FALSE;
											faultTimer.IN := FALSE;
                                        END_IF
									ELSIF faultTimer.Q THEN
										faultTimer.IN := FALSE;
										faults.failedToOpen.Trigger();
										state := PRESSURE_BAR_STATES.Fault;
                                    END_IF

    PRESSURE_BAR_STATES.JawOpened :            //Jaw is opened.  If in semi auto mode, go to close jaw after extend dwell.
                                    IF (semiAutoModeSelected AND startCyclePB) THEN
                                        timerExtendDwell.IN := TRUE;
                                    END_IF

                                    IF timerExtendDwell.Q OR (autoModeSelected AND _amCloseJaw) OR HMIData.pressureBarService.retractCommand THEN
                                        state := PRESSURE_BAR_STATES.CloseJaw;
                                        _amCloseJaw := FALSE;
										HMIData.pressureBarService.retractCommand := FALSE;
                                        timerExtendDwell.IN := FALSE;
                                    END_IF

    PRESSURE_BAR_STATES.CloseJaw :            //Close jaw by retracting cylinder
                                    RetractCylinder();
                                    state := PRESSURE_BAR_STATES.ClosingJaw;

    PRESSURE_BAR_STATES.ClosingJaw :            //
                                    //This delay is a debounce after the sensor is seen
                                    faultTimer.PT := T#3S;
									faultTimer.IN := TRUE;
									IF iPressureBarRetracted THEN
                                        timerRetractedDebounce.IN := TRUE;
                                        IF timerRetractedDebounce.Q THEN
                                            state := PRESSURE_BAR_STATES.JawClosed;
                                            timerRetractedDebounce.IN := FALSE;
											faultTimer.IN := FALSE;
                                        END_IF
									ELSIF faultTimer.Q THEN
										faultTimer.IN := FALSE;
										faults.failedToClose.Trigger();
										ExtendCylinderLowPressure();
										state := PRESSURE_BAR_STATES.Fault;
                                    END_IF
									IF NOT iPressureBarNotObstructed AND NOT iPressureBarRetracted THEN
										faults.obstructionDetected.Trigger();
										ExtendCylinderLowPressure();
										faultTimer.IN := FALSE;
										state := PRESSURE_BAR_STATES.Fault;
									END_IF

    PRESSURE_BAR_STATES.JawClosed :            //Go to sealing if seal bar enabled, otherwise if in auto mode go to open jaw after retract dwell. Else go back to idle

                                    IF (semiAutoModeSelected AND startCyclePB) THEN
                                        timerRetractDwell.IN := TRUE;
                                    END_IF
									IF iPressureBarNotObstructed THEN
										timerObsSwitchFault.IN := TRUE;
										IF timerObsSwitchFault.Q THEN
											ExtendCylinderLowPressure();
											faults.obstructionFailedToSwitch.Trigger();
											state := PRESSURE_BAR_STATES.Fault;
										END_IF
									ELSE
										timerObsSwitchFault.IN := FALSE;
									END_IF

                                    IF timerRetractDwell.Q OR (autoModeSelected AND _amOpenJaw) OR HMIData.pressureBarService.extendCommand THEN
                                        state := PRESSURE_BAR_STATES.OpenJaw;
										HMIData.pressureBarService.extendCommand := FALSE;
                                        _amOpenJaw := FALSE;
                                        timerRetractDwell.IN := FALSE;
                                    END_IF

    PRESSURE_BAR_STATES.Manual :    IF manualExhaustPB THEN
                                        ExhaustCylinder();
                                        manualExhaustPB := FALSE;
                                    ELSIF manualRetractPB THEN
                                        RetractCylinder();
                                        manualRetractPB := FALSE;
                                    ELSIF manualExtendHighPressurePB THEN
                                        ExtendCylinderHighPressure();
                                        manualExtendHighPressurePB := FALSE;
									ELSIF manualExtendLowPressurePB THEN
                                        ExtendCylinderLowPressure();
                                        manualExtendLowPressurePB := FALSE;
                                    END_IF

    PRESSURE_BAR_STATES.Fault :

END_CASE

IF NOT iPressureBarNotObstructed AND Globals.jawMovingIn THEN
										faults.obstructionDetected.Trigger();
										//ExtendCylinderLowPressure();
										ExhaustCylinder();
										faultTimer.IN := FALSE;
										state := PRESSURE_BAR_STATES.Fault;
END_IF
IF iPressureBarExtended AND iPressureBarRetracted THEN
	faults.sensorFault.Trigger();
END_IF

//Count cycles
incrementCount(CLK :=timerExtendDwell.Q);
IF incrementCount.Q THEN
    cumulativeHeadCycleCount := cumulativeHeadCycleCount + 1;
END_IF

METHOD AutoSealBag
VAR_INPUT
END_VAR

METHOD RetractCylinder
VAR_INPUT
END_VAR

oExtendCylinder := FALSE;
oRetractCylinder := TRUE;

METHOD AutoOpenJaw
VAR_INPUT
END_VAR

_amOpenJaw := TRUE;

METHOD ExhaustCylinder
VAR_INPUT
END_VAR

oExtendCylinder := FALSE;
oRetractCylinder := FALSE;

METHOD AutoDoneMovingPassthrough
VAR_INPUT
END_VAR

state := PRESSURE_BAR_STATES.Idle;

PROPERTY Mode : DEVICE_MODES

METHOD ExtendCylinderHighPressure
VAR_INPUT
END_VAR

oExtendCylinder := TRUE;
oRetractCylinder := FALSE;

PROPERTY Ready : BOOL

METHOD AutoCloseJaw
VAR_INPUT
END_VAR

_amCloseJaw := TRUE;

METHOD AutoMovingPassthrough
VAR_INPUT
END_VAR

//state := PRESSURE_BAR_STATES.Manual;
state := PRESSURE_BAR_STATES.Idle;

METHOD ExtendCylinderLowPressure
VAR_INPUT
END_VAR

oExtendCylinder := TRUE;
oRetractCylinder := TRUE;

(* ---- PRG_.st ---- *)
FUNCTION_BLOCK PRG_
VAR_INPUT
END_VAR
VAR_OUTPUT
END_VAR
VAR
END_VAR

(* ---- PrinterFB.st ---- *)
FUNCTION_BLOCK PrinterFB EXTENDS BaseComponentFB IMPLEMENTS IComponentStatus
VAR_INPUT
    autoSendLabel :BOOL;    // Automatically send a label
END_VAR
VAR_OUTPUT
    state : PRINTER_STATES;         // Printer State Machine
	oLowerPrintHead : BOOL;
	printHeadDebounced : BOOL;

END_VAR
VAR
    _amPrintNow : BOOL;                // Auto mode - print now
    _amSendPrintSignal : BOOL;        // Auto mode - send print signal
    _amGoToIdle : BOOL;                // Auto mode - Acked, go back to idle mode
    printHeadDebounce : TON;
    printHeadDebouneSetpoint : TIME := T#50MS;
    tcpServer : FB_TCPClient();
END_VAR

VAR_IN_OUT
END_VAR

//    Function Block: Printer
//    Description: This program manages the aspects of a (Zebra) printer
//    Created by: Ben Hess
//    Created Date: April 2nd, 2018
SUPER^();
// Enable TCP Server for label sending
tcpServer();

//Report as ready if mode is auto and we're not faulted
_ready := (_mode = DEVICE_MODES.Auto) AND NOT (state = PRINTER_STATES.Fault);

printHeadDebounce(PT:= printHeadDebouneSetpoint, Q=> printHeadDebounced);
IF enableONS.Q OR resetONS.Q THEN
    state := PRINTER_STATES.Idle;
	_reset := FALSE;
	_amGoToIdle := FALSE;
	_amSendPrintSignal := FALSE;
	_amPrintNow := FALSE;
END_IF

IF NOT enable THEN
    state := PRINTER_STATES.Fault;
	oRunPrinterRibbonUnwindMotor := FALSE;
	oLowerPrintHead := FALSE;
END_IF

//State machine for the printer
CASE state OF
    PRINTER_STATES.Idle :                            //Go to waiting for data if printer is ready
                                                    oRunPrinterRibbonUnwindMotor := FALSE;
													oPrinterStartPrint := FALSE;
													oLowerPrintHead := FALSE;
													printHeadDebounce.IN := FALSE;
													IF NOT printerDataReady THEN
                                                        IF autoSendLabel THEN
                                                            tcpServer.SendLabel();
                                                        END_IF
                                                        state := PRINTER_STATES.WaitingForData;
                                                    ELSE
                                                        state := PRINTER_STATES.DataReady;
                                                    END_IF

    PRINTER_STATES.WaitingForData :                    //If printerDataReady drops out the label data was received

                                                    IF printerDataReady THEN
                                                        state := PRINTER_STATES.DataReady;
                                                    END_IF

    PRINTER_STATES.DataReady :                        // Wait for command to begin printing
                                                    IF NOT printerDataReady THEN
														state := PRINTER_STATES.Idle;
													END_IF
													IF _mode = DEVICE_MODES.Auto AND _amPrintNow THEN
                                                        state := PRINTER_STATES.BeginPrintCycle;
                                                        _amPrintNow := FALSE;
                                                        oLowerPrintHead := TRUE;
                                                        oRunPrinterRibbonUnwindMotor := TRUE;
														//oPrinterStartPrint := TRUE;
                                                    END_IF

    PRINTER_STATES.BeginPrintCycle :                // Start printing

                                                    printHeadDebounce.IN := TRUE;
                                                    IF printHeadDebounce.Q AND _amSendPrintSignal THEN
                                                        oPrinterStartPrint := TRUE;
                                                        state := PRINTER_STATES.Printing;
                                                        printHeadDebounce.IN := FALSE;
                                                        _amSendPrintSignal := FALSE;
                                                    END_IF

    PRINTER_STATES.FeedAtPrintSpeed :                //

    PRINTER_STATES.Printing :                        //While printing, wait for End of Print signal
                                                    IF printerEndOfPrint THEN
                                                        oPrinterStartPrint := FALSE;
                                                        oLowerPrintHead := FALSE;

                                                        state := PRINTER_STATES.DonePrinting;
                                                    END_IF

    PRINTER_STATES.DonePrinting :                    //Done printing, feed a little more through
                                                    IF _mode = DEVICE_MODES.Auto AND _amGoToIdle THEN
                                                        oRunPrinterRibbonUnwindMotor := FALSE;
                                                        state := PRINTER_STATES.Idle;
                                                        _amGoToIdle := FALSE;
														HMIData.printerCycles.Increment();
														HMIData.printHeadClean.Increment();
                                                        Globals.printerCycleCounts := Globals.printerCycleCounts + 1;
                                                    END_IF

    PRINTER_STATES.FeedThrough :

    PRINTER_STATES.Ready :

    PRINTER_STATES.Fault :

END_CASE

METHOD AutoSendPrintSignal
VAR_INPUT
END_VAR

_amSendPrintSignal := TRUE;

PROPERTY Mode : DEVICE_MODES

PROPERTY Ready : BOOL

METHOD AutoPrintNow
VAR_INPUT
END_VAR

_amPrintNow := TRUE;

METHOD AutoAckPrintDone
VAR_INPUT
END_VAR
_amGoToIdle := TRUE;

(* ---- PrinterFB_Mode2.st ---- *)
FUNCTION_BLOCK PrinterFB_Mode2 EXTENDS BaseComponentFB IMPLEMENTS IComponentStatus
VAR_INPUT
    autoSendLabel :BOOL;    // Automatically send a label
	ribbonEncoderPulse : BOOL;	// Ribbon Encoder Input
	enableRibbonDetection : BOOL := TRUE;
END_VAR
VAR_OUTPUT
    state : PRINTER_STATES;         // Printer State Machine
	oLowerPrintHead : BOOL;
	printHeadDebounced : BOOL;
	ribbonFault : FB_Fault(name := 'Printer Ribbon Fault');
END_VAR
VAR
    _amPrintNow : BOOL;                // Auto mode - print now
    _amSendPrintSignal : BOOL;        // Auto mode - send print signal
    _amGoToIdle : BOOL;                // Auto mode - Acked, go back to idle mode
    printHeadDebounce : TON;
	printStarted : BOOL;
    printHeadDebouneSetpoint : TIME := T#50MS;
    tcpServer : FB_TCPClient();
	endOfPrintONS : Standard.F_TRIG();
	printerRibbonMovingTimer1 : Standard.TON;
	printerRibbonMovingTimer2 : Standard.TON;
	printerRibbonMovingSettleTime : TIME := T#450MS;
END_VAR

VAR_IN_OUT
END_VAR

//    Function Block: Printer
//    Description: This program manages the aspects of a (Zebra) printer
//    Created by: Ben Hess
//    Created Date: April 2nd, 2018
SUPER^();
// Enable TCP Server for label sending
tcpServer();
endOfPrintONS(CLK := printerEndOfPrint);
//Report as ready if mode is auto and we're not faulted
_ready := (_mode = DEVICE_MODES.Auto) AND NOT (state = PRINTER_STATES.Fault);

printerRibbonMovingTimer1(PT := printerRibbonMovingSettleTime);
printerRibbonMovingTimer2(PT := printerRibbonMovingSettleTime);

printHeadDebounce(PT:= printHeadDebouneSetpoint, Q=> printHeadDebounced);
printStarted := printerEndOfPrint;

IF enableONS.Q OR resetONS.Q THEN
    state := PRINTER_STATES.Idle;
	_reset := FALSE;
	_amGoToIdle := FALSE;
	_amSendPrintSignal := FALSE;
	_amPrintNow := FALSE;
	printHeadDebounced := FALSE;
	oRunPrinterRibbonUnwindMotor := FALSE;
	oLowerPrintHead := FALSE;
	printerRibbonMovingTimer1.IN := FALSE;
	printerRibbonMovingTimer2.IN := FALSE;
END_IF

IF NOT enable THEN
    state := PRINTER_STATES.Fault;
	oRunPrinterRibbonUnwindMotor := FALSE;
	oLowerPrintHead := FALSE;
END_IF

IF HMIData.printHeadServiceRaise THEN
	oLowerPrintHead := FALSE;
	HMIData.printHeadServiceRaise := FALSE;
ELSIF HMIData.printHeadServiceLower THEN
	oLowerPrintHead := TRUE;
	HMIData.printHeadServiceLower := FALSE;
END_IF

//State machine for the printer
CASE state OF
    PRINTER_STATES.Idle :                            //Go to waiting for data if printer is ready
                                                    oRunPrinterRibbonUnwindMotor := FALSE;
													oPrinterStartPrint := FALSE;
													printHeadDebounce.IN := FALSE;
													printHeadDebounced := FALSE;
													printerRibbonMovingTimer1.IN := FALSE;
													printerRibbonMovingTimer2.IN := FALSE;
													IF NOT printerDataReady THEN
                                                        IF autoSendLabel THEN
                                                            tcpServer.SendLabel();
                                                        END_IF
                                                        state := PRINTER_STATES.WaitingForData;
                                                    ELSE
                                                        state := PRINTER_STATES.DataReady;
                                                    END_IF

    PRINTER_STATES.WaitingForData :                    //If printerDataReady drops out the label data was received

                                                    IF printerDataReady THEN
                                                        state := PRINTER_STATES.DataReady;
                                                    END_IF

    PRINTER_STATES.DataReady :                        // Wait for command to begin printing
                                                    IF NOT printerDataReady THEN
														state := PRINTER_STATES.Idle;
													END_IF
													IF _mode = DEVICE_MODES.Auto AND _amPrintNow THEN
                                                        state := PRINTER_STATES.BeginPrintCycle;
                                                        _amPrintNow := FALSE;
														printHeadDebounce.IN := TRUE;
                                                        oLowerPrintHead := TRUE;
                                                        oRunPrinterRibbonUnwindMotor := TRUE;
														//oPrinterStartPrint := TRUE;
                                                    END_IF

    PRINTER_STATES.BeginPrintCycle :                // Start printing

                                                    IF _amSendPrintSignal THEN
                                                        oPrinterStartPrint := TRUE;

                                                        state := PRINTER_STATES.Printing;
                                                        printHeadDebounce.IN := FALSE;
                                                        _amSendPrintSignal := FALSE;
                                                    END_IF

    PRINTER_STATES.FeedAtPrintSpeed :                //

    PRINTER_STATES.Printing :                        //While printing, wait for End of Print signal
													printerRibbonMovingTimer1.IN := ribbonEncoderPulse;
													printerRibbonMovingTimer2.IN := NOT ribbonEncoderPulse;
                                                    IF endOfPrintONS.Q OR printerRibbonMovingTimer1.Q OR printerRibbonMovingTimer2.Q THEN
                                                        oPrinterStartPrint := FALSE;
                                                        oLowerPrintHead := FALSE;
														IF printerRibbonMovingTimer1.Q OR printerRibbonMovingTimer2.Q THEN
															ribbonFault.Trigger();
														END_IF
														printerRibbonMovingTimer1.IN := FALSE;
														printerRibbonMovingTimer2.IN := FALSE;

                                                        //oRunPrinterRibbonUnwindMotor := FALSE;
                                                        state := PRINTER_STATES.DonePrinting;
                                                    END_IF

    PRINTER_STATES.DonePrinting :                    //Done printing, feed a little more through
                                                    IF _mode = DEVICE_MODES.Auto AND _amGoToIdle THEN
                                                        oRunPrinterRibbonUnwindMotor := FALSE;
                                                        state := PRINTER_STATES.Idle;
                                                        _amGoToIdle := FALSE;
														HMIData.printerCycles.Increment();
														HMIData.printHeadClean.Increment();
                                                        Globals.printerCycleCounts := Globals.printerCycleCounts + 1;
                                                    END_IF

    PRINTER_STATES.FeedThrough :

    PRINTER_STATES.Ready :

    PRINTER_STATES.Fault :

END_CASE

METHOD AutoSendPrintSignal
VAR_INPUT
END_VAR

_amSendPrintSignal := TRUE;

METHOD AutoPrintNow
VAR_INPUT
END_VAR

_amPrintNow := TRUE;

METHOD AutoAckPrintDone
VAR_INPUT
END_VAR
_amGoToIdle := TRUE;

PROPERTY Mode : DEVICE_MODES

PROPERTY Ready : BOOL

(* ---- SerialMotorTestFB.st ---- *)
FUNCTION_BLOCK SerialMotorTestFB
VAR_INPUT
    runMotorPB : BOOL;
END_VAR
VAR_OUTPUT
END_VAR
VAR
    //testMotor : FB_AppliedMotionStepServoRTU();
    //orientalMotor : FB_OrientalAZDrive();
END_VAR

(*
orientalMotor(modbusInBuffer := OrientalMotorModbusRead,
                stepsPerInchSetpoint := 2122,
                reversePolarity := FALSE,
                operatingCurrentDefault := 100,
                modbusCommandOutBuffer := OrientalMotorCommandWrites,
                modbusParametersOutBuffer := OrientalMotorParameterWrites,
                triggerCommandWrite => OrientalMotorTriggerCommandWrite,
                triggerParameterWrite => OrientalMotorTriggerParameterWrite);
orientalMotor.Execute();
*)

IF runMotorPB THEN
    //testMotor.MoveDistance(12,100,100,215);
    //testMotor.HomeNow();

    //orientalMotor.MoveDistance(12,10000,10000,10000);
    runMotorPB := FALSE;
END_IF

(* ---- StepServoStatusFB.st ---- *)
FUNCTION_BLOCK StepServoStatusFB
VAR_INPUT
    statusCode : INT;
END_VAR
VAR_OUTPUT
    motorEnabled : BOOL;        //Motor Enabled (Motor Disabled if this bit = 0)
    sampling : BOOL;      //Sampling (for Quick Tuner)
    driveFaulted : BOOL;      //Drive Fault (check Alarm Code)
    inPosition : BOOL;      //In Position (motor is in position)
    moving : BOOL;      //Moving (motor is moving)
    jogging    : BOOL;      //Jogging (currently in jog mode)
    stopping : BOOL;      //Stopping (in the process of stopping from a stop command)
    waitingForInput : BOOL;      //Waiting (for an input; executing a WI command)
    saving : BOOL;      //Saving (parameter data is being saved)
    alarmPresent : BOOL;      //Alarm present (check Alarm Code)
    homing : BOOL;      //Homing (executing an SH command)
    waitingForTime : BOOL;      //Waiting (for time; executing a WD or WT command)
    wizardRunning : BOOL;      //Wizard running (Timing Wizard is running)
    checkingEncoder    : BOOL;      //Checking encoder (Timing Wizard is running)
    Q_ProgramRunning : BOOL;      //Q Program is running
    initializing : BOOL;      //Initializing (happens at power up) ; Servo Ready (for SV200 drives only)
END_VAR
VAR
END_VAR

//    Fucntion Block: StepServoStatus
//    Description: This unpacks the step servo status bits from the status word received over modbus
//    Created by: Ben Hess
//    Created Date: January 26th, 2018

motorEnabled := statusCode.0;
sampling := statusCode.1;
driveFaulted := statusCode.2;
inPosition := statusCode.3;
moving := statusCode.4;
jogging := statusCode.5;
stopping := statusCode.6;
waitingForInput    := statusCode.7;
saving := statusCode.8;
alarmPresent := statusCode.9;
homing := statusCode.10;
waitingForTime := statusCode.11;
wizardRunning := statusCode.12;
checkingEncoder := statusCode.13;
Q_ProgramRunning := statusCode.14;
initializing := statusCode.15;

(* ---- TimeLeftFB.st ---- *)
FUNCTION_BLOCK TimeLeftFB
VAR_INPUT
    targetDate : DATE_AND_TIME;
END_VAR
VAR_OUTPUT
    timeLeft : DATE_AND_TIME;

    targetMonths : UINT;
    targetDays : UINT;
    targetHours : UINT;
    targetMinutes : UINT;
    targetSeconds : UINT;
    currentMonths : UINT;
    currentDays : UINT;
    currentHours : UINT;
    currentMinutes : UINT;
    currentSeconds : UINT;
    timeLeftMonths : UINT;
    timeLeftDays : UINT;
    timeLeftHours : UINT;
    timeLeftMinutes : UINT;
    timeLeftSeconds : UINT;
    timeLeftString : STRING[250];
END_VAR
VAR
    iState                    : INT;
    udiUtcTime             : UDINT;
    udiUtcTimeLocal     : UDINT;
    strTimeDate         : SYSTIMEDATE;
    strTimeDateLocal     : SYSTIMEDATE;
    dtDateTimeUTC        : DATE_AND_TIME;
    timeLeftTime        : TIME;
    timeLeftDWORD        : DWORD;
    dDateUTC            : DATE;
    todTimeOfDayUTC        : TOD;

    tSysStartTime        : TIME;
    systimeStartNano    : SYSTIME;
    udiStartTimeResult    : UDINT;

    udiResult             : UDINT;

    GetDateAndTime            : DTU.GetDateAndTime;
    SetTimeZoneInformation    : DTU.SetTimeZoneInformation;

    dtCurrent                : DATE_AND_TIME;
    dtConcated                : DATE_AND_TIME;
    eWeekday                 : RTCLK.WEEKDAY;
    uiYear                     : UINT;
    uiMonth                     : UINT;
    uiDay                     : UINT;
    uiHour                     : UINT;
    uiMinute                 : UINT;
    uiSecond                 : UINT;

    dtuError                : DTU.ERROR;
END_VAR

CASE iState OF

    0:
        iState:= 1;

    1:  // retrieves the target date and time, including the timezone information which was set before
        GetDateAndTime( xExecute:= TRUE);
        IF GetDateAndTime.xDone THEN
            dtCurrent:= GetDateAndTime.dtDateAndTime;
            GetDateAndTime(xExecute:= FALSE);
            //timeLeft := TIME_TO_DT(DT_TO_TIME(targetDate) - DT_TO_TIME(dttarget));
            iState:= 2;
        END_IF
        IF GetDateAndTime.xError THEN
            GetDateAndTime(xExecute:= FALSE);
            iState:= 32767;
        END_IF

    2: (*set a spedific date and time --> returns a variable of type DATE_AND_TIME
         DateConcat --> set only date information --> returns a variable of type DATE
         TODConcat  --> set only the time information  --> returns a variable of TOD (Time of day) *)
        dtConcated := DTU.DTConcat(uiYear:= 2010, uiMonth:= 10, uiDay:= 5,
                            uiHour:= 9, uiMinute:= 20, uiSecond:= 12, peError:=ADR(dtuError));
        IF dtuError = 0 THEN
            iState := 3;
        ELSE
            iState := 32767;
        END_IF

    3:  (*a DATE_AND_TIME variable is splitted in its parts, like year, month, day etc.
            DateSplit --> the same function for a DATE variable
            TODSplit  --> the same function for a TOD variable *)
        dtuError := DTU.DTSplit(
            dtDateAndTime := dtCurrent,
            puiYear := ADR(uiYear),
            puiMonth := ADR(currentMonths),
            puiDay := ADR(currentDays),
            puiHour := ADR(currentHours),
            puiMinute := ADR(currentMinutes),
            puiSecond := ADR(currentSeconds));
        dtuError := DTU.DTSplit(
            dtDateAndTime := targetDate,
            puiYear := ADR(uiYear),
            puiMonth := ADR(targetMonths),
            puiDay := ADR(targetDays),
            puiHour := ADR(targetHours),
            puiMinute := ADR(targetMinutes),
            puiSecond := ADR(targetSeconds));

        IF dtuError = 0 THEN
            iState:= 1;
        ELSE
            iState:= 32767;
        END_IF

    32767: ; //error

END_CASE

timeLeftMonths := currentMonths - targetMonths;
timeLeftDays := currentDays - targetDays;
timeLeftHours := currentHours - targetHours;
timeLeftMinutes := currentMinutes - targetMinutes;
timeLeftSeconds := currentSeconds - targetSeconds;

timeLeftString := CONCAT('Time left to PMMI: ', UINT_TO_STRING(timeLeftMonths));
timeLeftString := CONCAT(' Months, ', UINT_TO_STRING(timeLeftDays));
timeLeftString := CONCAT(' Days, ', UINT_TO_STRING(timeLeftHours));
timeLeftString := CONCAT(' Hours, ', UINT_TO_STRING(timeLeftMinutes));
timeLeftString := CONCAT(' Minutes, ', UINT_TO_STRING(timeLeftSeconds));
timeLeftString := CONCAT(' Seconds', '');

timeLeftDWORD := DT_TO_DWORD(targetDate) - DT_TO_DWORD(dtCurrent);
timeLeftDays := DWORD_TO_UINT(timeLeftDWORD / 86000);

(* ---- Faults.st ---- *)
PROGRAM Faults
VAR
	reverseFault : FB_HMIFault;
END_VAR

reverseFault(refFault := PRG_Bagger.moabHead.bagDelivery.reverseFault);

(* ---- PRG_Bagger.st ---- *)
PROGRAM PRG_Bagger
VAR_INPUT

END_VAR
VAR_OUTPUT

END_VAR
VAR
    moabHead : FB_MOABHead;
    //angledHead : FB_20degHead();
    //pneuHead : FB_PneumaticHead();
    testEIPMotor : FB_AppliedMotionStepServoEIPBase();
    faultHandler : FB_FaultHandler();
	hmiInitiate : BOOL;
	msfMotorFaults : ARRAY[0..100] OF MotorCommFault;
	numberOfMSFFaults : UINT;
	msfCommFaultONS : R_TRIG();
	msfFaultListFull : BOOL;
	festoFaults : ARRAY[0..100] OF MotorCommFault;
	numberOfFestoFaults : UINT;
	festoCommFaultONS : R_TRIG();
	festoFaultListFull : BOOL;
	currentDateAndTime : GetTime();
	resetCommFaults : BOOL;
	i : INT;
	reverseFault : FB_HMIFault := (refFault := PRG_Bagger.moabHead.bagDelivery.reverseFault);
	faultActiveONS : FB_ONS;
END_VAR

//    Program: PRG_Bagger
//    Description: This program glues together the whole machine and all of its components.
//
//    Created by: Ben Hess
//    Created Date: Tuesday, April 17, 2018

moabHead();
//pneuHead();
faultHandler();
hmiInitiate := HMIData.initiateCycle;
currentDateAndTime();
//msfCommFaultONS(CLK := MSFMotor.xDiagnosticAvailable);
HMIData.bagEdgePhotoeyeCovered := NOT iBagNotPresent;
oSoftStart := TRUE;

HMIData.airFilterClean();
HMIData.pressureBarGuideShaftGuides();
HMIData.driveRollerClean();
HMIData.printHeadClean();
HMIData.pressureBarLeak(iExtended := iPressureBarExtended, iRetracted := iPressureBarRetracted, maximumStrokeTime := (TO_REAL(HMIData.passthroughSetting / 26.6)) + 0.3);
HMIData.loadPlateLeak(iExtended := iLoadPlateExtended, iRetracted := iLoadPlateRetracted, maximumStrokeTime := 0.4);
//HMIData.msfHorizontalMotorTemp(iDriveTemp := sealFlattenerHorizontalMotorInputs[4]);
//HMIData.bagDeliveryMotorTemp(iDriveTemp := bagDeliveryMotorInputs[4]);
//HMIData.passthroughMotorTemp(iDriveTemp := jawPasstrhoughMotorInputs[4]);

IF resetCommFaults THEN
	FOR i := 0 TO numberOfMSFFaults BY 1 DO
		msfMotorFaults[i].message := '';
		msfMotorFaults[i].timeOfFault := DT#1970-1-1-1:0:0;
	END_FOR
	numberOfMSFFaults := 0;
	msfFaultListFull := FALSE;
	resetCommFaults := FALSE;
END_IF

//HMIData.version := SVN_VERSION_INFO.VERSION;

HMIData.faultActive := GlobalObjects.CollectionOfActiveFaults.faultActive;
faultActiveONS(CLK := GlobalObjects.CollectionOfActiveFaults.faultActive);
IF faultActiveONS.OSR THEN
	moabHead.hmiLight.TurnOff();
END_IF

(* ---- PRG_MainProgram.st ---- *)
PROGRAM PRG_MainProgram
VAR
    incrementSolenoidCounter1 : R_TRIG();
    incrementSolenoidCounter2 : R_TRIG();
    incrementSolenoidFailedCounter2 : R_TRIG();
    GripperCycleCount : DINT; //Gripper Cycle Counter
    runPrinterPB : BOOL;
    cycleTimeMax : TIME;
    cycleTimeMaxDINT : DINT;
    ctfb : OSCAT_BASIC.CYCLE_TIME();
    profileThis :BOOL;
    solenoidState1 : SOLENOID_TEST_STATES;
    solenoidState2 : SOLENOID_TEST_STATES;
    getTimeTilPMMI : TimeLeftFB();
	displayPassthroughChangeDistance : REAL;
	displayPassthroughChangeDistance2 : REAL;
	checkSolenoid2ExtendTimer : TON := (PT := T#100MS);
	checkedSolenoid2Status : BOOL;
	firstScanDone : BOOL;
	printDeltaTimer : TON := (PT := T#5S);
	lastPrinterDelta : TIME;
	endPrintOSF : Standard.R_TRIG;
	CSVWriter : FB_WriteToFile() := (xFilePath := 'C:/printerDelta.csv');
	stringToLog : STRING;
	testWrite : BOOL;
	hmiLight : FB_HMILight;
	versionInfo : VERSION;
END_VAR
//    Program: Main (PLC_PRG)
//    Description: This program serves as a base for the MOAB Prototype
//    Created by: Ben Hess
//    Created Date: January 16th, 2018

endPrintOSF(CLK := printerEndOfPrint);
printDeltaTimer(IN := oPrinterStartPrint);
// IF endPrintOSF.Q OR testWrite THEN
// 	lastPrinterDelta := printDeltaTimer.ET;
// 	Globals.lastPrinterDelta := printDeltaTimer.ET;
// 	stringToLog :=  CONCAT(TO_STRING(PRG_Bagger.currentDateAndTime.dtCurrent),',');
// 	stringToLog := Standard.CONCAT(stringToLog,TO_STRING(printDeltaTimer.ET));
// 	CSVWriter.xText_Write := stringToLog;
// 	CSVWriter.xWrite := TRUE;
// 	testWrite := FALSE;
// END_IF
//
// CSVWriter(
// 	xFilePath:= ,
// 	xText_Write:= ,
// 	xAppend_OverWrite:= TRUE,
// 	xAppend_Pos:= ,
// 	xWrite:= ,
// 	xRead:= ,
// 	xLine_No_To_Read:= ,
// 	xText_Read=> ,
// 	xDone=> );
// IF CSVWriter.xDone THEN
// 	CSVWriter.xWrite := FALSE;
// END_IF

ctfb(ct_max => cycleTimeMax);
cycleTimeMaxDINT := TIME_TO_DINT(cycleTimeMax);
profileThis := TIME_TO_DINT(ctfb.ct_last) >= 25;
// Run other programs
//PRG_PneumaticHead();
PRG_Bagger();
Faults();
versionInfo := GetVersion();
HMIData.version := Standard.CONCAT(TO_STRING(versionInfo.uiMajor),'.');
	BPLog.AppendToString(ADR(HMIData.version), CONCAT(TO_STRING(versionInfo.uiMinor),'.'));
	BPLog.AppendToString(ADR(HMIData.version), CONCAT(TO_STRING(versionInfo.uiServicePack),'.'));
	BPLog.AppendToString(ADR(HMIData.version), TO_STRING(versionInfo.uiPatch));
	//BPLog.AppendToString(ADR(HMIData.version), TO_STRING(GetTextProperty("VersionPostfix")));
IF NOT firstScanDone THEN
	GlobalObjects.CollectionOfLoggable.RegisterAll(internalLogger := Globals.SystemLog);
	GlobalObjects.CollectionOfInitialzable.InitializeAll();
	firstScanDone := TRUE;
	// After first scan turn off flag set by StartDone system event
	Globals.firstScan := FALSE;
END_IF

// Start executing objects that implement IExecuteAutomatically
IF firstScanDone THEN
	GlobalObjects.CollectionOfExecutable.ExecuteAll();
	Globals.SystemLog();
END_IF

IF HMIData.ackAllFaults THEN
	GlobalObjects.CollectionOfActiveFaults.AckAll();
	HMIData.ackAllFaults := FALSE;
END_IF

getTimeTilPMMI(targetDate := DT#2018-10-14-8:0:0);

//First scan flag is set by task handler and reset in main routine here
IF Globals.firstScan THEN
    Globals.firstScan := FALSE;
END_IF

displayPassthroughChangeDistance := (UDINT_TO_REAL(Globals.passthroughChangeDistance) / 10);
displayPassthroughChangeDistance2 := (UDINT_TO_REAL(Globals.passthroughChangeDistance2) / 10.0);
